FUNCTION_BLOCK FB_MergingFiFo
//FB_MergingFiFo 
//
VAR_INPUT
	FunctionNumber  : E_FunctionNumber;
	Disable			: BOOL; 	// Make this E_Function disabled, ie PriorityControl will not return this E_FunctionNumber
	CompareNextFunc	: E_FunctionNumber; // Check if next is set to this function. F_BEGIN_FUNCTION = No check performed		  
END_VAR

VAR_OUTPUT
	ePrevFunctionNumber		: E_FunctionNumber;		//the function number that has the highest priority to enter into Loop or intersection.	  
END_VAR
VAR CONSTANT 
    ELEMENTLAST 	: INT:=20;
	ELEMENTFIRST	: INT:=1;
	STARTZONE		: INT:=1;
	EmptyBuffer		: ST_FifoBuffer:= (eFunctionNumber:=0,EntryOK:=0, Occupied:=0) ; 
END_VAR 
VAR	
	_Buffer					: ARRAY[ELEMENTFIRST..ELEMENTLAST] OF ST_FifoBuffer;	
END_VAR
VAR_TEMP
	i						: INT;
END_VAR


ePrevFunctionNumber :=E_FunctionNumber.F_BEGIN_FUNCTION;

_M_AddItem(FunctionNumber,Disable);

//return the first item in the list (that are not disabled)
//Check if function is occupied, iterate entire buffer array
FOR i:=ELEMENTFIRST TO ELEMENTLAST BY 1 DO
	IF(_Buffer[i].EntryOK AND _Buffer[i].Occupied) THEN
		ePrevFunctionNumber :=_Buffer[i].eFunctionNumber;						
		EXIT;
	END_IF
END_FOR

METHOD PRIVATE _M_AddItem : BOOL  //FIFO table
VAR_INPUT
	FunctionNumber  : E_FunctionNumber;
	Disable			: BOOL; 	// Make this E_Function disabled, ie PriorityControl will not return this E_FunctionNumber		
END_VAR

VAR	
	myBufferIx		: INT:=0;		
	i:INT;
	j:INT;
	
END_VAR

//search for function in buffer, get myBufferIx
FOR myBufferIx := ELEMENTFIRST TO ELEMENTLAST BY 1 DO
	IF(_Buffer[myBufferIx].eFunctionNumber=FunctionNumber) THEN EXIT; END_IF
END_FOR

//if entry was not already in buffer -> search for first empty slot
IF(myBufferIx>ELEMENTLAST) THEN // no item found	
	FOR myBufferIx := ELEMENTFIRST TO ELEMENTLAST BY 1 DO
		IF(_Buffer[myBufferIx].eFunctionNumber=0) THEN EXIT;	END_IF
	END_FOR
END_IF

//if no emtpy slot was found, then buffer full, so return.
IF(myBufferIx>ELEMENTLAST) THEN RETURN; END_IF

//------------------------------------------------------------------------
// By now, the Buffer Ix is determined
// Add function number to the buffer list
//------------------------------------------------------------------------
_Buffer[myBufferIx].eFunctionNumber := FunctionNumber;
_Buffer[myBufferIx].EntryOK := NOT Disable AND _M_EntryOk(FunctionNumber);

//------------------------------------------------------------------------
// Check all functions in the list being occupied
// Check if functions being occupied
//------------------------------------------------------------------------

IF(_Buffer[myBufferIx].eFunctionNumber>0) THEN
	_Buffer[myBufferIx].Occupied:=FALSE;		
	_Buffer[myBufferIx].Occupied:=_M_Enabled(_Buffer[myBufferIx].eFunctionNumber); //check occupied and handover enabled.
	IF( NOT _Buffer[myBufferIx].Occupied) THEN
		//Clear buffer
		_Buffer[myBufferIx]:=EmptyBuffer;			
	END_IF
END_IF

//------------------------------------------------------------------------
// Sort items, 
//------------------------------------------------------------------------

_M_SortFifo();
	
_M_AddItem := TRUE;
END_METHOD

METHOD PRIVATE _M_Enabled : BOOL
VAR_INPUT
	FunctionNumber : E_FunctionNumber; 
END_VAR
VAR
	rZoneData		:REFERENCE TO ST_ZoneData;
	rZoneTrspEnable :REFERENCE TO ST_TransportEnable;	
	i:INT;
	Tu_index :DINT;
END_VAR


IF( NOT __ISVALIDREF(FunctionRegistry[FunctionNumber].rFunction)) THEN RETURN; END_IF
IF( NOT __ISVALIDREF(FunctionRegistry[FunctionNumber].rFunctionInterface)) THEN RETURN; END_IF

FOR i:=STARTZONE TO NUMBER_OF_ZONES_PER_FUNCTION BY 1 DO
	rZoneData REF= FunctionRegistry[FunctionNumber].rFunction.ZoneData[i];
	rZoneTrspEnable REF=FunctionRegistry[FunctionNumber].rFunction.ZoneInterface[i].In.Enable;	

	_M_Enabled:= _M_Enabled OR	F_PB_GetTransportControlDataRef(FunctionNumber,i).Occupied OR F_PB_GetTransportControlDataRef(FunctionNumber,i).DataPresent;
	
	IF NOT (rZoneData.AddOn.Orders.Enable AND rZoneData.AddOn.Orders.EnableHandover AND rZoneTrspEnable.HandOver AND rZoneTrspEnable.Transport) THEN
		_M_Enabled :=FALSE;
		EXIT;
	END_IF
	
	Tu_index := F_PB_GetTransportControlDataRef(FunctionNumber,i).TU_DataIndex;
	IF(Tu_index>0) THEN
		IF(NOT TU_Table.TU_DataTable[Tu_index].DataSet.JobPresent) THEN
			_M_Enabled :=FALSE;
			EXIT;
		END_IF
	END_IF
			
	//check if handover was completed, then remove from buffer
	IF(F_PB_GetTransportControlDataRef(FunctionNumber,i).eHandOverState= E_HandOverState.COMPLETE) THEN
		_M_Enabled :=FALSE;
		EXIT;
	END_IF
		
	
END_FOR
END_METHOD

METHOD PRIVATE _M_EntryOk : BOOL
VAR_INPUT
	FunctionNumber : E_FunctionNumber;	
END_VAR
VAR
	rZoneData		:REFERENCE TO ST_ZoneData;
	rZoneTrspEnable :REFERENCE TO ST_TransportEnable;
	i:INT;
	ElementNumber	: E_ElementNumber;
END_VAR
_M_EntryOk :=FALSE;
IF( NOT __ISVALIDREF(FunctionRegistry[FunctionNumber].rFunction)) THEN RETURN; END_IF
IF( NOT __ISVALIDREF(FunctionRegistry[FunctionNumber].rFunctionInterface)) THEN RETURN; END_IF
IF( NOT __ISVALIDREF(FunctionRegistry[FunctionNumber].rFunctionData)) THEN RETURN; END_IF
IF( NOT __ISVALIDREF(FunctionRegistry[FunctionNumber].rSettingsFunction)) THEN RETURN; END_IF

//check that there are no active errors in element, functon or zones

ElementNumber := FunctionRegistry[FunctionNumber].rSettingsFunction.eElementLink;
IF(__ISVALIDREF(ElementRegistry[ElementNumber].rElementData))THEN
	IF( NOT ElementRegistry[ElementNumber].rElementData.ErrorData.FunctionErrorPending AND 
		ElementRegistry[ElementNumber].rElementData.ErrorData.ErrorState <> E_ErrorState.ERROR) THEN
		_M_EntryOk :=TRUE;
	END_IF	
END_IF	



// check if element/function is started
_M_EntryOk := _M_EntryOk AND FunctionRegistry[FunctionNumber].rFunctionInterface.In.Element.OperationState.eState = E_PositionState.STARTED;								
//check if any zone/Function/element is disabled
_M_EntryOk := _M_EntryOk AND F_CheckAllEnabled(FunctionNumber);

//check that input function also has next defined (Should point to DTU but is not checked!!)
IF(THIS^.CompareNextFunc>E_FunctionNumber.F_BEGIN_FUNCTION AND FunctionRegistry[FunctionNumber].rFunctionInterface.In.eNextFunctionNumber<>CompareNextFunc) THEN
	_M_EntryOk := FALSE;
END_IF
END_METHOD

METHOD PRIVATE _M_SortFiFo : BOOL
VAR_INPUT
END_VAR
VAR
	i,j:INT;
END_VAR
FOR i:=ELEMENTFIRST TO ELEMENTLAST-1 BY 1 DO	
	IF(_Buffer[i].eFunctionNumber=0) THEN
		FOR j:=i+1 TO ELEMENTLAST BY 1 DO
			IF(_Buffer[j].eFunctionNumber <> 0) THEN
				_Buffer[i] := _Buffer[j];
				_Buffer[j] := EmptyBuffer;				
				EXIT;
			END_IF
		END_FOR
		EXIT;	//No need iterate over entire buffer. this will be covered next cycle.
	END_IF	
END_FOR
END_METHOD

METHOD PUBLIC M_GetFifoIndex : E_FunctionNumber
VAR_INPUT
	Index:INT; // 1 is the most prioritized Function
END_VAR
VAR
	myIndex,ix,i:INT;	
END_VAR

IF(Index<ELEMENTFIRST) THEN
	myIndex:= ELEMENTFIRST;
ELSIF(Index>ELEMENTLAST) THEN
	myIndex:= ELEMENTLAST;
ELSE
	myIndex:=Index;
END_IF


//return the first item in the list (that are not disabled)
//Check if function is occupied, iterate all zones
FOR i:=ELEMENTFIRST TO ELEMENTLAST BY 1 DO
	IF(_Buffer[i].EntryOK AND _Buffer[i].Occupied) THEN
		ix:= ix+1;
		IF(ix=myIndex) THEN
			M_GetFifoIndex :=_Buffer[i].eFunctionNumber;
			EXIT;
		END_IF			
	END_IF
END_FOR
END_METHOD

//Set function to the lowest priority, ie move to last positoin in FIFO
METHOD PUBLIC M_MoveToLast : BOOL
VAR_INPUT
	FunctionNumber : E_FunctionNumber;
	//Index:INT;	
END_VAR
VAR
	i:INT;
	MyIndex:Int;
END_VAR
IF(FunctionNumber=0) THEN RETURN; END_IF

//return the first item in the list (that are not disabled)
//Check if function is occupied, iterate all zones
FOR i:=ELEMENTFIRST TO ELEMENTLAST BY 1 DO
	IF(_Buffer[i].eFunctionNumber = FunctionNumber) THEN
		//Clear buffer -> remove from FIFO-> it will be added next cycle
		_Buffer[i]:=EmptyBuffer;
		EXIT;				
	END_IF
END_FOR

//sort fifo (_M_SortFiFo()) not needed, this will be carried out when re-adding the unit
END_METHOD

END_FUNCTION_BLOCK

(* stored: Version 1.1.0.1, ProductVersion 3.1.4024.9
   POU FB_MergingFiFo: Id {4286b1cd-f58d-4a0b-8a3d-de5baac41ba3}, SpecialFunc None
   Method _M_AddItem: Id {414e55fd-95d5-4b24-88b5-fb77b974e0c2}
   Method _M_Enabled: Id {4cda8fe9-1d8c-4afb-8213-acc908c9602e}
   Method _M_EntryOk: Id {b79a8ca9-ace9-4627-8411-17c223bb4215}
   Method _M_SortFiFo: Id {9b8d0123-bc61-4652-abe3-c3fc6717b5b4}
   Method M_GetFifoIndex: Id {aa951cb5-170f-4fe1-950b-c2b206e98fce}
   Method M_MoveToLast: Id {ec69daa9-41de-4241-9c8b-24bc6ad8385e} *)
